{attribute 'qualified_only'}
VAR_GLOBAL
	
	{attribute 'S7.Out'}
	{attribute 'S7.Address' := 'db2.dbx0.0'}
	imAlive : BOOL;
	{attribute 'S7.In'}
	{attribute 'S7.Address' := 'db2.dbx1.0'}
	otherSystemAlive :BOOL;
	
	{attribute 'S7.Out'}
	{attribute 'S7.Address' := 'db2.int2'}
	counter : INT;
	
END_VAR

(* stored: Version 1.1.0.1, ProductVersion 3.1.4024.3
   GVL GVL: Id {cb2e065a-2489-42d8-9dbd-7260f7cbc0ae} *)
